// TwinCAT 3 PLC project ExercisePWM
// ProgramVersion: 3.1.4024.0
// libraries:
//   Tc2_Standard, * (Beckhoff Automation GmbH)
//   Tc2_System, * (Beckhoff Automation GmbH)
//   Tc3_Module, * (Beckhoff Automation GmbH)
// project tree:
//   / PlcTask.TcTTO
//   POUs/ FB_PWM.TcPOU, MAIN.TcPOU
// (motion and I/O tree: see PLC project checkerfunctions)
// real-time tasks:
//   TASK PlcTask: cycle T#10ms, priority 20, ADS port 350
//   TASK PlcTask1: cycle T#10ms, priority 21, ADS port 351
//   TASK PlcTask2: cycle T#10ms, priority 22, ADS port 352
//   TASK PlcTask3: cycle T#10ms, priority 23, ADS port 353
//   TASK PlcTask4: cycle T#10ms, priority 24, ADS port 354
//   TASK PlcTask5: cycle T#10ms, priority 25, ADS port 355
//   TASK PlcTask6: cycle T#10ms, priority 26, ADS port 356
//   TASK PlcTask7: cycle T#10ms, priority 27, ADS port 357

CONFIGURATION ExercisePWM
    RESOURCE PLC ON TwinCAT3
        TASK PlcTask(INTERVAL := T#10ms, PRIORITY := 21);
        PROGRAM MAIN WITH PlcTask : MAIN;
    END_RESOURCE
END_CONFIGURATION

// ---- POUs/MAIN.TcPOU
PROGRAM MAIN
VAR
pwmInstance : FB_PWM;
END_VAR

pwmInstance(fPeriod := 1000, fDutyCycle := 50); // Voorbeeldwaarden

END_PROGRAM

// ---- POUs/FB_PWM.TcPOU
FUNCTION_BLOCK FB_PWM
VAR_INPUT
    fPeriod    : REAL;    // Periode van het PWM-signaal in ms
    fDutyCycle : REAL;    // Duty cycle in procenten
END_VAR
VAR_OUTPUT
    bPWMOutput : BOOL;    // PWM output
END_VAR
VAR
    tTimer     : TON;     // Timer voor het PWM-signaal
END_VAR

// PWM-logica
tTimer(IN := tTimer.Q, PT := TO_TIME(fPeriod));
IF tTimer.ET < TO_TIME(fPeriod * fDutyCycle / 100) THEN
    bPWMOutput := TRUE;
ELSE
    bPWMOutput := FALSE;
END_IF

END_FUNCTION_BLOCK
